PROGRAM MAIN
VAR
END_VAR

END_PROGRAM

(* stored: Version 1.1.0.1
   POU MAIN: Id {32814a16-c380-41c7-a0cd-38aa00ddda83} *)
